// Struckig
// Copyright (C) 2022 Stefan Besler

// This program is free software: you can redistribute it and/or modify
// it under the terms of the GNU General Public License as published by
// the Free Software Foundation, either version 3 of the License, or
// (at your option) any later version.

// This program is distributed in the hope that it will be useful,
// but WITHOUT ANY WARRANTY; without even the implied warranty of
// MERCHANTABILITY or FITNESS FOR A PARTICULAR PURPOSE.  See the
// GNU General Public License for more details.
//
// You should have received a copy of the GNU General Public License
// along with THIS PROGRAM.  IF NOT, see <http://www.gnu.org/licenses/>.
TYPE INTERNAL Block :
STRUCT
  Pmin : ProfileDesc; // Save min Profile so that it doesn't need to be recalculated in Step2
  Tmin : LREAL; // [s]
  A, B : BlockInterval; // Max. 2 intervals can be blocked: called a and b with corresponding profiles, order does not matter  
END_STRUCT
END_TYPE

(* stored: Version 1.1.0.1
   DUT Block: Id {4be6a195-68c0-418b-ad15-0b28c6e2cb63} *)
